// TIA Portal V17 export
// export: Created 2024-09-27T18:53:42.8437049Z, ExportSetting WithDefaults, DisplayName Totally Integrated Automation Portal, DisplayVersion V17, DisplayName TIA Portal Openness, DisplayVersion V17, DisplayName TIA Portal Version Control Interface, DisplayVersion V17, DisplayName STEP 7 Professional, DisplayVersion V17, DisplayName STEP 7 Safety, DisplayVersion V17, DisplayName WinCC Professional, DisplayVersion V17
FUNCTION "MANUAL" : Void   // FC1, LAD
{ S7_Optimized_Access := 'TRUE' }
VERSION : 0.1
// stored: AutoNumber true, IsIECCheckEnabled false, SetENOAutomatically false, UDAEnableTagReadback false
   VAR_TEMP   // added for the SCL form of the ladder/FBD networks
      _w1 : Bool;
   END_VAR
BEGIN

REGION Network 1: WARUNKI DLA TRYBU RĘCZNEGO
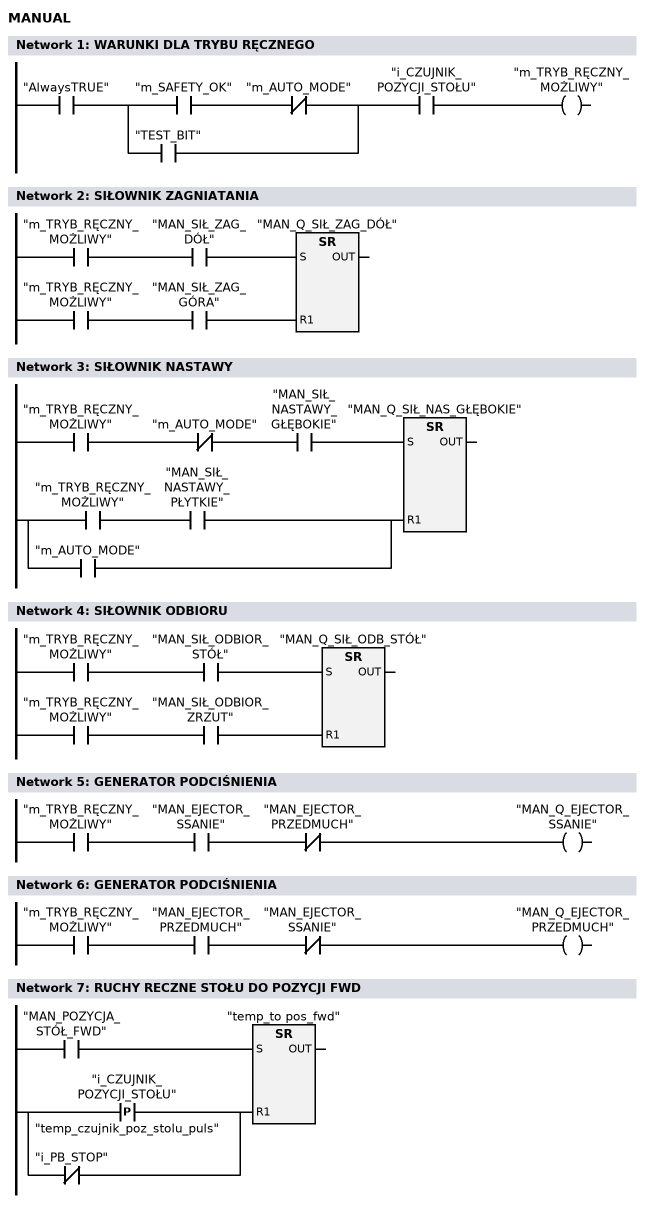
   RUNG wire#powerrail
      Contact( "AlwaysTRUE" )
      wire#w1
      Contact( "m_SAFETY_OK" )
      I_Contact( "m_AUTO_MODE" )
      wire#w2
      Contact( "i_CZUJNIK_POZYCJI_STOŁU" )
      Coil( "m_TRYB_RĘCZNY_MOŻLIWY" )
   END_RUNG
   RUNG wire#w1
      Contact( "TEST_BIT" )
   END_RUNG wire#w2
   // the same network as SCL:
   "m_TRYB_RĘCZNY_MOŻLIWY" := "AlwaysTRUE" AND (("m_SAFETY_OK" AND NOT "m_AUTO_MODE") OR "TEST_BIT") AND "i_CZUJNIK_POZYCJI_STOŁU";
END_REGION

REGION Network 2: SIŁOWNIK ZAGNIATANIA
   RUNG wire#powerrail
      Contact( "m_TRYB_RĘCZNY_MOŻLIWY" )
      Contact( "MAN_SIŁ_ZAG_DÓŁ" )
      S_SR(operand := "MAN_Q_SIŁ_ZAG_DÓŁ", r1 := wire#w1)
   END_RUNG
   RUNG wire#powerrail
      Contact( "m_TRYB_RĘCZNY_MOŻLIWY" )
      Contact( "MAN_SIŁ_ZAG_GÓRA" )
   END_RUNG wire#w1
   // the same network as SCL:
   IF "m_TRYB_RĘCZNY_MOŻLIWY" AND "MAN_SIŁ_ZAG_DÓŁ" THEN
       "MAN_Q_SIŁ_ZAG_DÓŁ" := TRUE;   // SR flip-flop
   END_IF;
   IF "m_TRYB_RĘCZNY_MOŻLIWY" AND "MAN_SIŁ_ZAG_GÓRA" THEN "MAN_Q_SIŁ_ZAG_DÓŁ" := FALSE; END_IF;
END_REGION

REGION Network 3: SIŁOWNIK NASTAWY
   RUNG wire#powerrail
      Contact( "m_TRYB_RĘCZNY_MOŻLIWY" )
      I_Contact( "m_AUTO_MODE" )
      Contact( "MAN_SIŁ_NASTAWY_GŁĘBOKIE" )
      S_SR(operand := "MAN_Q_SIŁ_NAS_GŁĘBOKIE", r1 := wire#w1)
   END_RUNG
   RUNG wire#powerrail
      Contact( "m_TRYB_RĘCZNY_MOŻLIWY" )
      Contact( "MAN_SIŁ_NASTAWY_PŁYTKIE" )
   END_RUNG wire#w1
   RUNG wire#powerrail
      Contact( "m_AUTO_MODE" )
   END_RUNG wire#w1
   // the same network as SCL:
   IF "m_TRYB_RĘCZNY_MOŻLIWY" AND NOT "m_AUTO_MODE" AND "MAN_SIŁ_NASTAWY_GŁĘBOKIE" THEN
       "MAN_Q_SIŁ_NAS_GŁĘBOKIE" := TRUE;   // SR flip-flop
   END_IF;
   IF ("m_TRYB_RĘCZNY_MOŻLIWY" AND "MAN_SIŁ_NASTAWY_PŁYTKIE") OR "m_AUTO_MODE" THEN
       "MAN_Q_SIŁ_NAS_GŁĘBOKIE" := FALSE;
   END_IF;
END_REGION

REGION Network 4: SIŁOWNIK ODBIORU
   RUNG wire#powerrail
      Contact( "m_TRYB_RĘCZNY_MOŻLIWY" )
      Contact( "MAN_SIŁ_ODBIOR_STÓŁ" )
      S_SR(operand := "MAN_Q_SIŁ_ODB_STÓŁ", r1 := wire#w1)
   END_RUNG
   RUNG wire#powerrail
      Contact( "m_TRYB_RĘCZNY_MOŻLIWY" )
      Contact( "MAN_SIŁ_ODBIOR_ZRZUT" )
   END_RUNG wire#w1
   // the same network as SCL:
   IF "m_TRYB_RĘCZNY_MOŻLIWY" AND "MAN_SIŁ_ODBIOR_STÓŁ" THEN
       "MAN_Q_SIŁ_ODB_STÓŁ" := TRUE;   // SR flip-flop
   END_IF;
   IF "m_TRYB_RĘCZNY_MOŻLIWY" AND "MAN_SIŁ_ODBIOR_ZRZUT" THEN "MAN_Q_SIŁ_ODB_STÓŁ" := FALSE; END_IF;
END_REGION

REGION Network 5: GENERATOR PODCIŚNIENIA
   RUNG wire#powerrail
      Contact( "m_TRYB_RĘCZNY_MOŻLIWY" )
      Contact( "MAN_EJECTOR_SSANIE" )
      I_Contact( "MAN_EJECTOR_PRZEDMUCH" )
      Coil( "MAN_Q_EJECTOR_SSANIE" )
   END_RUNG
   // the same network as SCL:
   "MAN_Q_EJECTOR_SSANIE" := "m_TRYB_RĘCZNY_MOŻLIWY" AND "MAN_EJECTOR_SSANIE" AND NOT "MAN_EJECTOR_PRZEDMUCH";
END_REGION

REGION Network 6: GENERATOR PODCIŚNIENIA
   RUNG wire#powerrail
      Contact( "m_TRYB_RĘCZNY_MOŻLIWY" )
      Contact( "MAN_EJECTOR_PRZEDMUCH" )
      I_Contact( "MAN_EJECTOR_SSANIE" )
      Coil( "MAN_Q_EJECTOR_PRZEDMUCH" )
   END_RUNG
   // the same network as SCL:
   "MAN_Q_EJECTOR_PRZEDMUCH" := "m_TRYB_RĘCZNY_MOŻLIWY" AND "MAN_EJECTOR_PRZEDMUCH" AND NOT "MAN_EJECTOR_SSANIE";
END_REGION

REGION Network 7: RUCHY RECZNE STOŁU DO POZYCJI FWD
   RUNG wire#powerrail
      Contact( "MAN_POZYCJA_STÓŁ_FWD" )
      S_SR(operand := "temp_to pos_fwd", r1 := wire#w1)
   END_RUNG
   RUNG wire#powerrail
      P_Contact(operand := "i_CZUJNIK_POZYCJI_STOŁU", bit := "temp_czujnik_poz_stolu_puls")
   END_RUNG wire#w1
   RUNG wire#powerrail
      I_Contact( "i_PB_STOP" )
   END_RUNG wire#w1
   // the same network as SCL:
   #_w1 := "i_CZUJNIK_POZYCJI_STOŁU" AND NOT "temp_czujnik_poz_stolu_puls";   // rising edge of "i_CZUJNIK_POZYCJI_STOŁU"
   "temp_czujnik_poz_stolu_puls" := "i_CZUJNIK_POZYCJI_STOŁU";
   IF "MAN_POZYCJA_STÓŁ_FWD" THEN
       "temp_to pos_fwd" := TRUE;   // SR flip-flop
   END_IF;
   IF #_w1 OR NOT "i_PB_STOP" THEN "temp_to pos_fwd" := FALSE; END_IF;
END_REGION
END_FUNCTION
